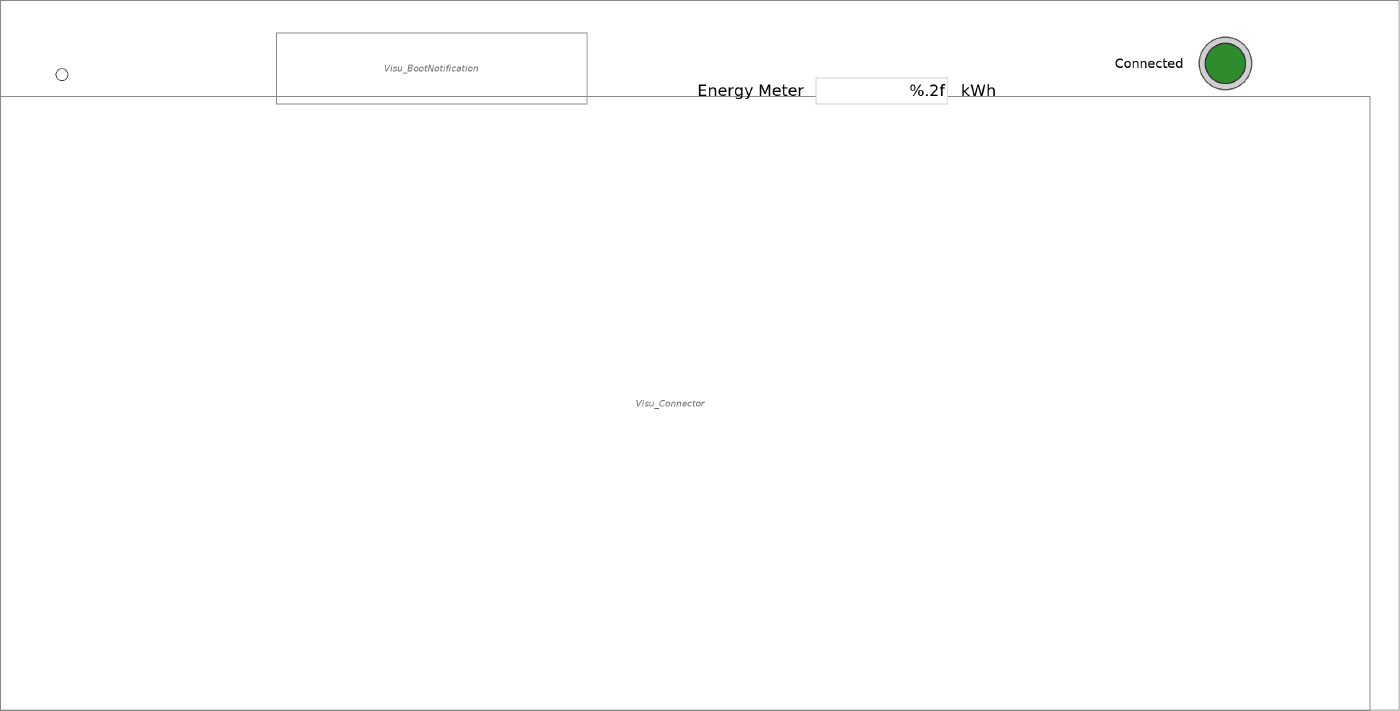
VISUALIZATION Visu_Station  // 1588x807
VAR_IN_OUT
	fbStation 		: FB_Station;
END_VAR
VAR 
	nConnectorVisu :UDINT; 
END_VAR
    Frame (-34,109 1588x698), frame switch variable: nConnectorVisu
        shows Visu_Connector(stConnector := fbStation._stVisu.aConnector[1], fbMeasurand := fbStation.arrMeasurands[1], bRemoteStart := fbStation._arrRemoteStart[1], bRemoteStop := fbStation._arrRemoteStop[1])
        shows Visu_Connector(stConnector := fbStation._stVisu.aConnector[2], fbMeasurand := fbStation.arrMeasurands[2], bRemoteStart := fbStation._arrRemoteStart[2], bRemoteStop := fbStation._arrRemoteStop[2])
    Frame (313,37 353x81)
        shows Visu_BootNotification(fbStation := fbStation)
    RadioButton (61,51 150x67), variable: nConnectorVisu
        Areas[0]: Text=Connector 1
        Areas[1]: Text=Connector 2
    Lamp1 (1355,37 70x70), variable: fbStation.bOpen, style: Lamp-Lamp1-Green
    Label (1184,37 161x70), "Connected"
    Textfield (925,88 150x30), "%.2f", text variable: fbStation.arrMeasurands[1].fEnergyActiveImportRegister + fbStation.arrMeasurands[2].fEnergyActiveImportRegister
    Label (765,88 150x30), "Energy Meter"
    Label (1079,88 62x30), "kWh"
END_VISUALIZATION

(* stored: Version 1.1.0.1
   Visu Visu_Station: Id {fdd06ce5-822a-42ef-b4bb-45e6db9ef96e} *)
